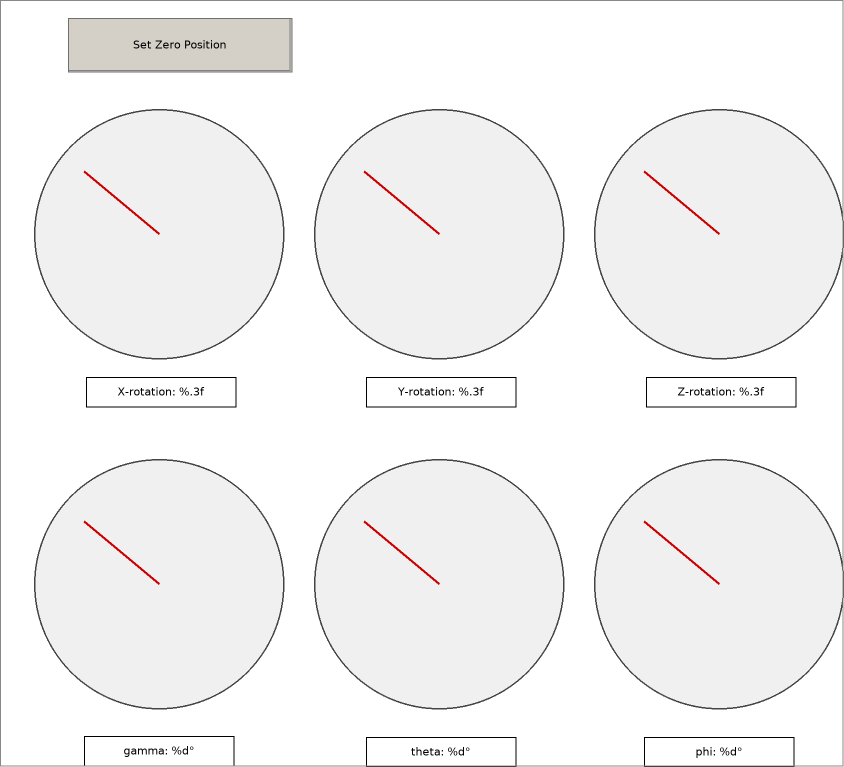
VISUALIZATION Visu  // 844x767
    Meter360 (34,109 250x250), value: MAIN.DegMovingHead[2], style: Meter-Meter360-Gray, scale format: %d, scale 0..360
    Rectangle (86,377 150x30), "X-rotation: %.3f", text variable: MAIN.Deg[0]
    Button (68,18 224x54), "Set Zero Position", colour toggle: MAIN.bReady
        p573394764: 16#FF80FF80
        p2175578022: 16#FF808080
        tap MAIN.bResetVisu
    Meter360 (314,109 250x250), value: MAIN.DegMovingHead[1], style: Meter-Meter360-Gray, scale format: %d, scale 0..360
    Rectangle (366,377 150x30), "Y-rotation: %.3f", text variable: MAIN.Deg[1]
    Meter360 (594,109 250x250), value: MAIN.DegMovingHead[0], style: Meter-Meter360-Gray, scale format: %d, scale 0..360
    Rectangle (646,377 150x30), "Z-rotation: %.3f", text variable: MAIN.Deg[0]
    Meter360 (34,459 250x250), value: MAIN.degGamma, style: Meter-Meter360-Gray, scale format: %d, scale 0..360
    Meter360 (314,459 250x250), value: MAIN.degTheta, style: Meter-Meter360-Gray, scale format: %d, scale 0..360
    Meter360 (594,459 250x250), value: MAIN.degPhi, style: Meter-Meter360-Gray, scale format: %d, scale 0..360
    Rectangle (84,736 150x30), "gamma: %d°", text variable: MAIN.degGamma
    Rectangle (366,737 150x30), "theta: %d°", text variable: MAIN.degTheta
    Rectangle (644,737 150x30), "phi: %d°", text variable: MAIN.degPhi
END_VISUALIZATION

(* stored: Version 1.1.0.1, ProductVersion 3.1.4024.12
   Visu Visu: Id {f35f0869-482b-4aa9-ae39-fc06821ab620} *)
